{attribute 'qualified_only'}
{attribute 'strict'}
TYPE MedewerkerToestand :
(
	wachtenOpKlant := 0,
	klantHelpen,
	verfMengen,
	verfGeven
);
END_TYPE

(* stored: Version 1.1.0.1, ProductVersion 3.1.4024.15
   DUT MedewerkerToestand: Id {5bbf5d48-5f6e-4895-b267-cd102d6f9319} *)
